Staubli VAL3: cmdResetAll.pgx

public program cmdResetAll(num x_nAxNum)
begin
  //复位所有信号
  doFaultReset[x_nAxNum]=false
  doEnableOp[x_nAxNum]=false
  doSwitchOn[x_nAxNum]=false
  doEnableVoltage[x_nAxNum]=false
  doQuickStop[x_nAxNum]=false
  delay(0.1)
end
